{attribute 'qualified_only'}
VAR_GLOBAL
	fvXref  : LREAL; // Toolpoint cartesian velocity. From joistick. Used for inv. vel kin and calculate path for pos controller
	fvYref  : LREAL;
	fvZref  : LREAL;
	fq4Dotref : LREAL; //Actuator angular velocity from inverse vel kinematics m/s
	f_q1_ref : LREAL; //Ref angles from inverse position kinematics radians
	f_q2_ref : LREAL;
	f_q3_ref : LREAL;
	bKinematicsSucsessful : BOOL;
END_VAR

(* stored: Version 1.1.0.1, ProductVersion 3.1.4024.12
   GVL G_InverseKinematics: Id {64159996-3342-42b4-9865-0a5dc597079d} *)
